FUNCTION_BLOCK SequenceTryout EXTENDS TcoCore.TcoSequencer
VAR
    counter : INT;
END_VAR
VAR
    //    eSequenceTest : E_SequenceTest := E_SequenceTest.WaitForStart;
    eSequenceTest : stSequenceTest;
    itfValveA     : I_DualPositionActuator := valveA;
    //~
    valveA : FB_DualPositionActuator
    (
        tActivateTimeout                     := T#3S
        , tDisableTimeout                    := T#3S
        , bIsActiveFeedbackSensorAvailable   := TRUE
        , bIsDisabledFeedbackSensorAvailable := TRUE
        , bNormallyDisabled                  := TRUE
    );
    //~
END_VAR
VAR CONSTANT
    simV : INT := 4;
END_VAR

(*~
    <docu>
        <summary>
            Main method of the sequener. Custom code needs to be placed here. The sequencer is executed by call of InstanceName.Run() method.
            This method is abstract, and it must be overridden in derived block.
        </summary>
    </docu>
~*)
METHOD PROTECTED Main : BOOL
counter := counter + 1;

IF (Step(eSequenceTest.WaitForStart, TRUE, 'Restore und Start')) THEN
    //    eSequenceTest := stSequenceTest.OpenValveAandB;
    StepCompleteWhen(counter MOD simV = 0);
END_IF

IF (Step(eSequenceTest.OpenValveAandB, TRUE, 'Zweiter Step')) THEN
    StepCompleteWhen(counter MOD simV = 0);
END_IF

IF (Step(999, TRUE, 'SEQUENCE COMPLETE')) THEN
    //--------------------------------------------
    CompleteSequence();
    //--------------------------------------------
END_IF;

IF (step(909, TRUE, 'ERROR Handling')) THEN
    ;
END_IF
END_METHOD

(*~
    <docu>
        <summary>
            This method is executed upon step completion.
            This method can be overridden in derived block by custom logic.
        </summary>
    </docu>
~*)
METHOD PROTECTED OnStepCompleted
counter := 1;
END_METHOD

END_FUNCTION_BLOCK

(* stored: Version 1.1.0.1, ProductVersion 3.1.4024.12
   POU SequenceTryout: Id {860826b7-16a6-49c4-a25c-c43416650a53}, SpecialFunc None
   Method Main: Id {52eba5f4-2f85-0df9-2be3-e03e48009737}
   Method OnStepCompleted: Id {91171987-4419-0888-30a1-a01a8d0ab40b} *)
